(* Schneider Machine Expert - Basic project Sala de metrologia 174.3-2026 alteracao set umidade, file version 2.7.0.0 *)
(* CompanyInformations: Name=Kaefer - Mercedes Benz - Delma, PhoneNumber=11975904673, Street=RUA ALFRED JURZYKOWSKI 56, City=SÃO BERNARDO DO CAMPO, ZipCode=09680-900, State=SÃO PAULO, Country=BRASIL, WebSite=MERCEDES BENZ *)
(* ProjectInformations: Name=CLP DE CONTROLE METROLOGIA 21, Description=SUBSTITUIÇÃO DO CLP SPYDER PUB4024S DA FABRICANTE HONEYWELL COM AVÁRIA POR OUTRO DA FABRICANTE SCHNEIDER:

MODELO DA CPU: TM221ME 16T/MG COM EXPANSÃO DE SAIDA ANÁLOGICA: TM3AQ2 COM DUAS SAIDA ANÁLOGICAS;

O PROJETO CONSISTE EM MANTER A TEMPERATURA EM 19.5°C a 20.8°C E UMIDADE 45 A 55% *)

HARDWARE
  Cpu 0: TM221ME16T/G
  ModuleExtensionObject 0: TM3AQ2/G
  EthernetConfiguration: NetworkName=M221, IpAllocationMode=FixedAddress, IpAddress=192.168.1.5, SubnetMask=255.255.255.0
  SerialLineConfiguration: Baud=Baud19200, Parity=ParityEven, DataBits=DataBits8, StopBits=StopBits1, PhysicalMedium=PhysicalMediumRs485, TransmissionMode=TransmissionModeModbusRtu, SlaveId=1, Addressing=SlaveAddressing
  MastTask: UsePeriodScanMode=false, PeriodScan=100
  FastTask: Period=255
  CpuBehavior: StartingMode=StartAsPreviousState, AutoSaveRamOnEeprom=true, WatchdogPeriod=250

SYMBOLS  (address, symbol, comment, settings)
  %M0       HABILITA_GERAL_  "Memoria de habilita geral"
  %M1       COMP_1_LIGAR_  "habilita compressor 1"
  %M2       LIGA_COMP_2  "habilita compressor 2"
  %M4       LIGA_VENTILAÇÃO
  %M5       STATUS_VENT_LIGA
  %M6       HABILITA_AQUEC
  %M8       FOTO_CELULA
  %S6       SB_TB1S  "Base de tempo de 1 s gerada por um relógio interno"
  %I0.0       "Habilita geral"
  %I0.1     TERMOSTATO_DE_SEG
  %I0.2     STATUS_VENT
  %I0.3     CHAVE_DE_FLUXO_
  %I0.4     PRESSOSTATO
  %Q0.0     VENTILADOR_LIGA_DESLIGA
  %Q0.1     COMPRESSOR_1__LIGADO_
  %Q0.2     COMP_2_LIGAR_
  %Q0.3     LIGA_UMIDIFICAÇÃO_
  %Q0.4     INIBIÇÃO_AQUECIMENTO
  %IW0.0      [Type=Type_0_10V, Scope=Scope_Normal, Minimum=0, Maximum=1000]
  %IW0.1      [Type=Type_0_10V, Scope=Scope_Normal, Minimum=0, Maximum=1000]
  %QW1.0      [Type=Type_0_10V, Scope=Scope_Customized, Minimum=0, Maximum=10000]

POU Novo POU
  (* SectionNumber=1 *)

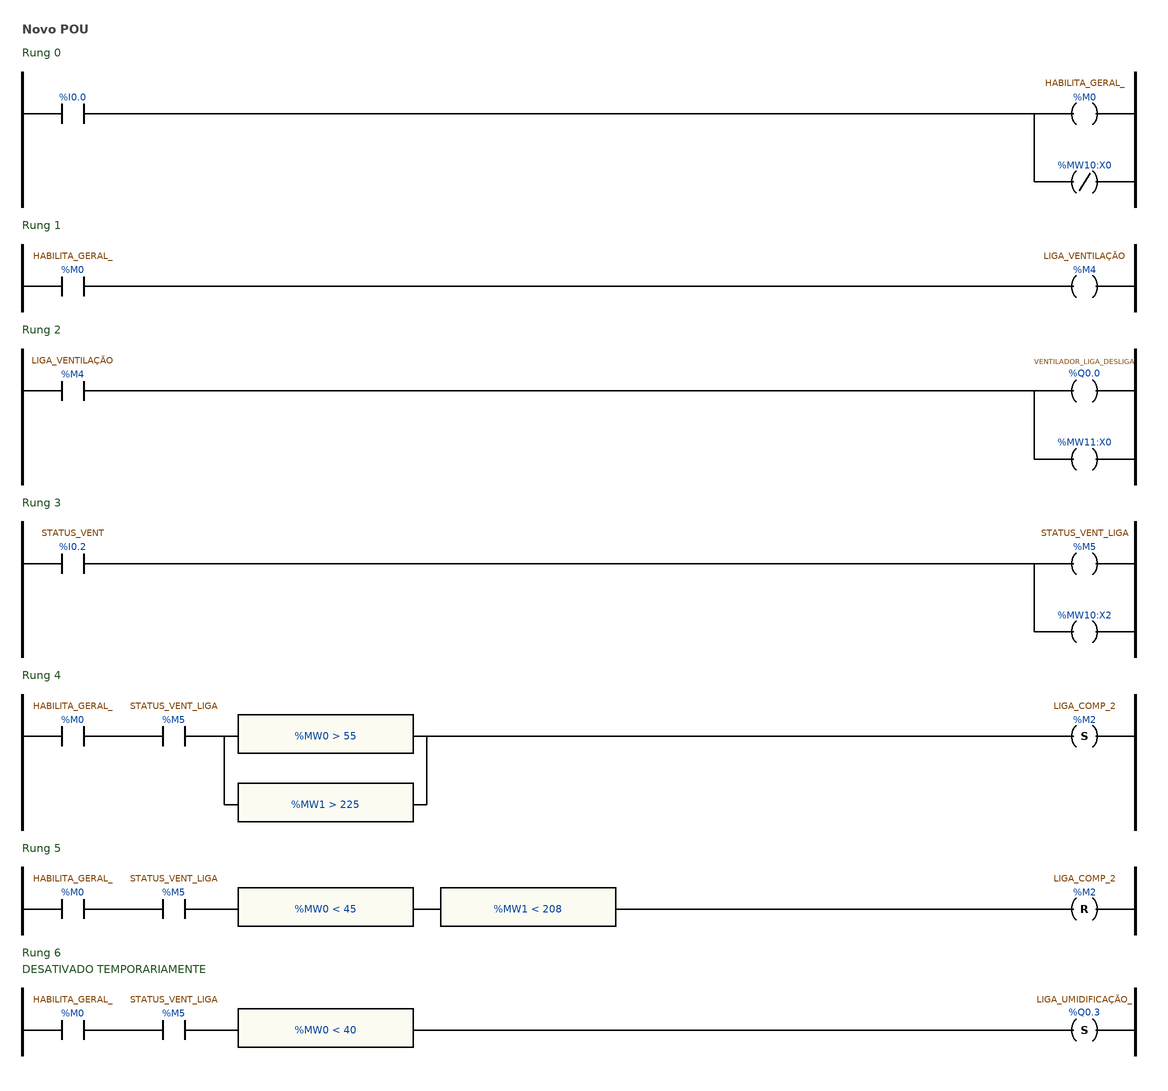

// Rung 0
  LD %I0.0
  ST %M0                  (* HABILITA_GERAL_ *)
  STN %MW10:X0
  // as ST:
  //   HABILITA_GERAL_ := %I0.0;
  //   %MW10:X0 := NOT %I0.0;

// Rung 1
  LD %M0                  (* HABILITA_GERAL_ *)
  ST %M4                  (* LIGA_VENTILAÇÃO *)
  // as ST:
  //   LIGA_VENTILAÇÃO := HABILITA_GERAL_;

// Rung 2
  LD %M4                  (* LIGA_VENTILAÇÃO *)
  ST %Q0.0                (* VENTILADOR_LIGA_DESLIGA *)
  ST %MW11:X0
  // as ST:
  //   VENTILADOR_LIGA_DESLIGA := LIGA_VENTILAÇÃO;
  //   %MW11:X0 := LIGA_VENTILAÇÃO;

// Rung 3
  LD %I0.2                (* STATUS_VENT *)
  ST %M5                  (* STATUS_VENT_LIGA *)
  ST %MW10:X2
  // as ST:
  //   STATUS_VENT_LIGA := STATUS_VENT;
  //   %MW10:X2 := STATUS_VENT;

// Rung 4
  LD %M0                  (* HABILITA_GERAL_ *)
  AND %M5                 (* STATUS_VENT_LIGA *)
  AND( [ %MW0 > 55 ]
  OR [ %MW1 > 225 ]
  )
  S %M2                   (* LIGA_COMP_2 *)
  // as ST:
  //   IF HABILITA_GERAL_ AND STATUS_VENT_LIGA AND (%MW0 > 55 OR %MW1 > 225) THEN LIGA_COMP_2 := TRUE; END_IF;

// Rung 5
  LD %M0                  (* HABILITA_GERAL_ *)
  AND %M5                 (* STATUS_VENT_LIGA *)
  AND [ %MW0 < 45 ]
  AND [ %MW1 < 208 ]
  R %M2                   (* LIGA_COMP_2 *)
  // as ST:
  //   IF HABILITA_GERAL_ AND STATUS_VENT_LIGA AND %MW0 < 45 AND %MW1 < 208 THEN LIGA_COMP_2 := FALSE; END_IF;

// Rung 6
// DESATIVADO TEMPORARIAMENTE
  LD %M0                  (* HABILITA_GERAL_ *)
  AND %M5                 (* STATUS_VENT_LIGA *)
  AND [ %MW0 < 40 ]
  S %Q0.3                 (* LIGA_UMIDIFICAÇÃO_ *)
  // as ST:
  //   IF HABILITA_GERAL_ AND STATUS_VENT_LIGA AND %MW0 < 40 THEN LIGA_UMIDIFICAÇÃO_ := TRUE; END_IF;

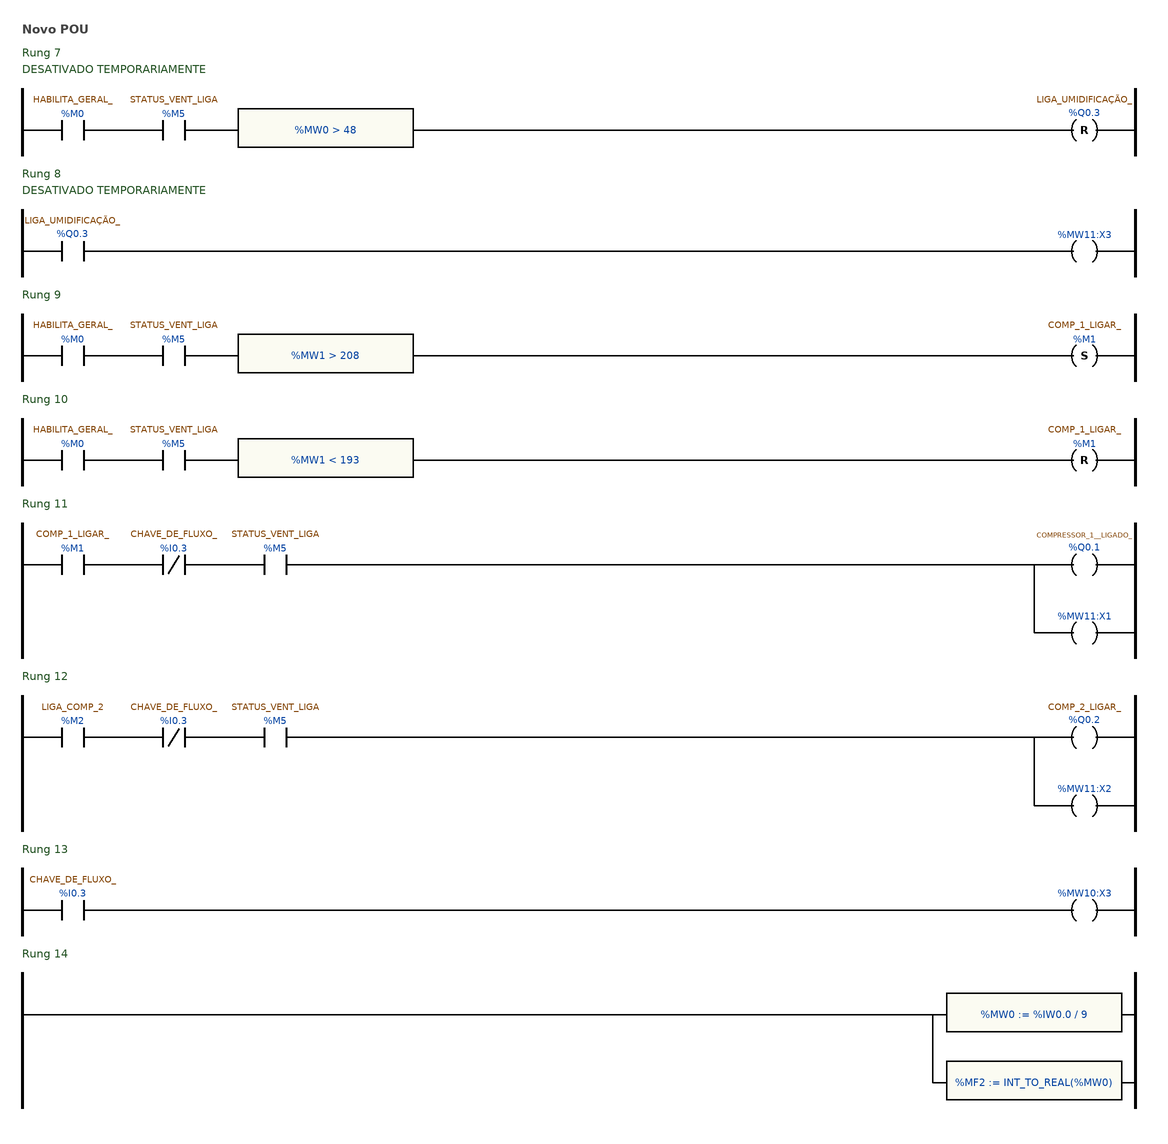

// Rung 7
// DESATIVADO TEMPORARIAMENTE
  LD %M0                  (* HABILITA_GERAL_ *)
  AND %M5                 (* STATUS_VENT_LIGA *)
  AND [ %MW0 > 48 ]
  R %Q0.3                 (* LIGA_UMIDIFICAÇÃO_ *)
  // as ST:
  //   IF HABILITA_GERAL_ AND STATUS_VENT_LIGA AND %MW0 > 48 THEN LIGA_UMIDIFICAÇÃO_ := FALSE; END_IF;

// Rung 8
// DESATIVADO TEMPORARIAMENTE
  LD %Q0.3                (* LIGA_UMIDIFICAÇÃO_ *)
  ST %MW11:X3
  // as ST:
  //   %MW11:X3 := LIGA_UMIDIFICAÇÃO_;

// Rung 9
  LD %M0                  (* HABILITA_GERAL_ *)
  AND %M5                 (* STATUS_VENT_LIGA *)
  AND [ %MW1 > 208 ]
  S %M1                   (* COMP_1_LIGAR_ *)
  // as ST:
  //   IF HABILITA_GERAL_ AND STATUS_VENT_LIGA AND %MW1 > 208 THEN COMP_1_LIGAR_ := TRUE; END_IF;

// Rung 10
  LD %M0                  (* HABILITA_GERAL_ *)
  AND %M5                 (* STATUS_VENT_LIGA *)
  AND [ %MW1 < 193 ]
  R %M1                   (* COMP_1_LIGAR_ *)
  // as ST:
  //   IF HABILITA_GERAL_ AND STATUS_VENT_LIGA AND %MW1 < 193 THEN COMP_1_LIGAR_ := FALSE; END_IF;

// Rung 11
  LD %M1                  (* COMP_1_LIGAR_ *)
  ANDN %I0.3              (* CHAVE_DE_FLUXO_ *)
  AND %M5                 (* STATUS_VENT_LIGA *)
  ST %Q0.1                (* COMPRESSOR_1__LIGADO_ *)
  ST %MW11:X1
  // as ST:
  //   COMPRESSOR_1__LIGADO_ := COMP_1_LIGAR_ AND NOT CHAVE_DE_FLUXO_ AND STATUS_VENT_LIGA;
  //   %MW11:X1 := COMP_1_LIGAR_ AND NOT CHAVE_DE_FLUXO_ AND STATUS_VENT_LIGA;

// Rung 12
  LD %M2                  (* LIGA_COMP_2 *)
  ANDN %I0.3              (* CHAVE_DE_FLUXO_ *)
  AND %M5                 (* STATUS_VENT_LIGA *)
  ST %Q0.2                (* COMP_2_LIGAR_ *)
  ST %MW11:X2
  // as ST:
  //   COMP_2_LIGAR_ := LIGA_COMP_2 AND NOT CHAVE_DE_FLUXO_ AND STATUS_VENT_LIGA;
  //   %MW11:X2 := LIGA_COMP_2 AND NOT CHAVE_DE_FLUXO_ AND STATUS_VENT_LIGA;

// Rung 13
  LD %I0.3                (* CHAVE_DE_FLUXO_ *)
  ST %MW10:X3
  // as ST:
  //   %MW10:X3 := CHAVE_DE_FLUXO_;

// Rung 14
  LD 1
  [ %MW0 := %IW0.0 / 9 ]
  [ %MF2 := INT_TO_REAL ( %MW0 ) ]
  // as ST:
  //   %MW0 := %IW0.0 / 9;
  //   %MF2 := INT_TO_REAL ( %MW0 );

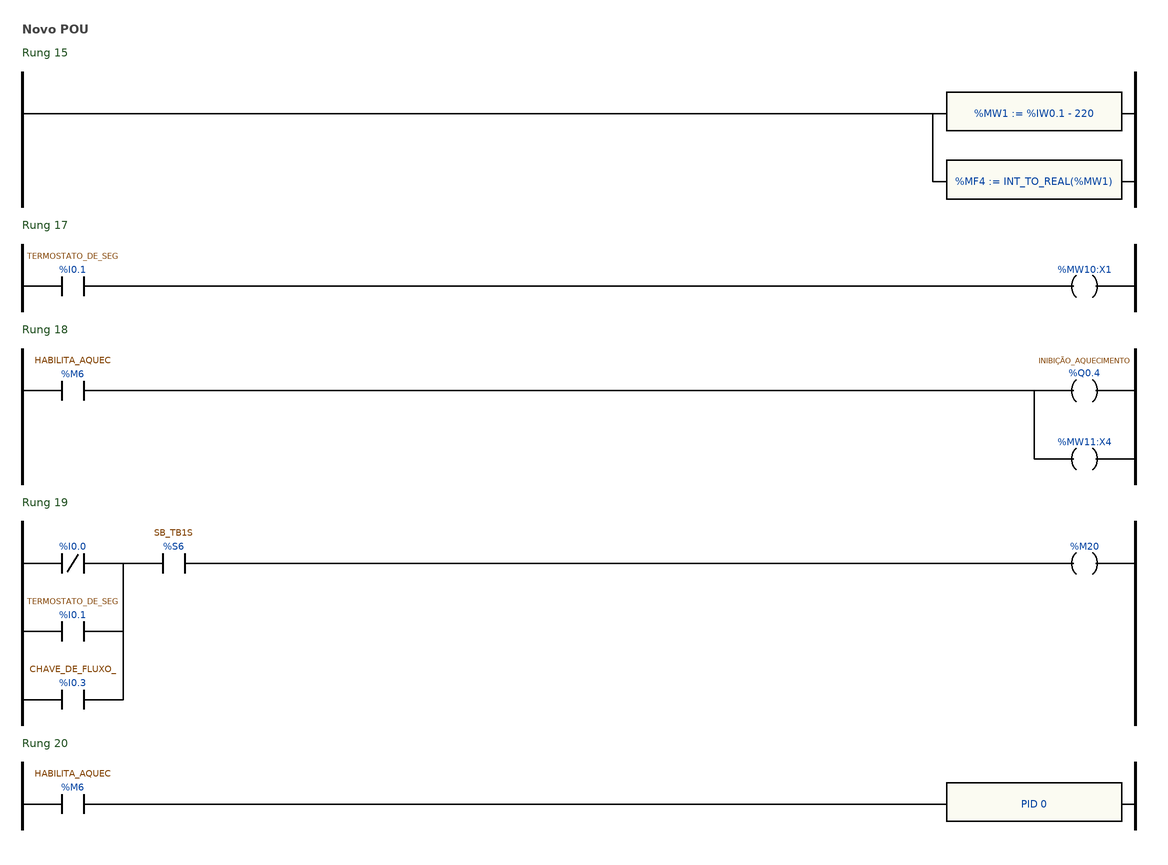

// Rung 15
  LD 1
  [ %MW1 := %IW0.1 - 220 ]
  [ %MF4 := INT_TO_REAL ( %MW1 ) ]
  // as ST:
  //   %MW1 := %IW0.1 - 220;
  //   %MF4 := INT_TO_REAL ( %MW1 );

// Rung 16
  LD %M5                  (* STATUS_VENT_LIGA *)
  ANDN %I0.1              (* TERMOSTATO_DE_SEG *)
  ANDN %I0.3              (* CHAVE_DE_FLUXO_ *)
  AND [ %MW1 > 225 ]
  ST %M6                  (* HABILITA_AQUEC *)
  // as ST:
  //   HABILITA_AQUEC := STATUS_VENT_LIGA AND NOT TERMOSTATO_DE_SEG AND NOT CHAVE_DE_FLUXO_ AND %MW1 > 225;
  (* the ladder stored for this rung does not match its IL; not drawn *)

// Rung 17
  LD %I0.1                (* TERMOSTATO_DE_SEG *)
  ST %MW10:X1
  // as ST:
  //   %MW10:X1 := TERMOSTATO_DE_SEG;

// Rung 18
  LD %M6                  (* HABILITA_AQUEC *)
  ST %Q0.4                (* INIBIÇÃO_AQUECIMENTO *)
  ST %MW11:X4
  // as ST:
  //   INIBIÇÃO_AQUECIMENTO := HABILITA_AQUEC;
  //   %MW11:X4 := HABILITA_AQUEC;

// Rung 19
  LDN %I0.0
  OR %I0.1                (* TERMOSTATO_DE_SEG *)
  OR %I0.3                (* CHAVE_DE_FLUXO_ *)
  AND %S6                 (* SB_TB1S *)
  ST %M20
  // as ST:
  //   %M20 := (NOT %I0.0 OR TERMOSTATO_DE_SEG OR CHAVE_DE_FLUXO_) AND SB_TB1S;

// Rung 20
  LD %M6                  (* HABILITA_AQUEC *)
  [ PID 0 ]
  // as ST:
  //   IF HABILITA_AQUEC THEN PID 0; END_IF;

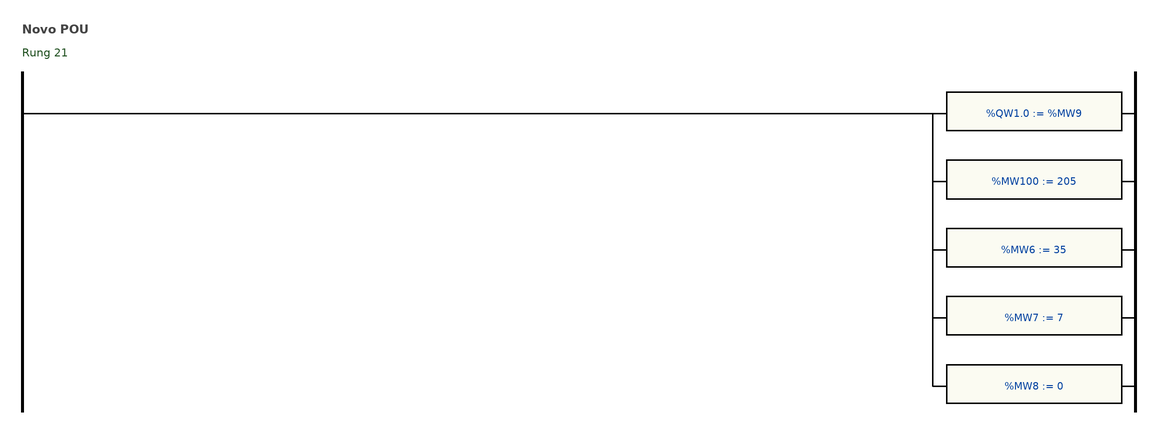

// Rung 21
  LD 1
  [ %QW1.0 := %MW9 ]
  [ %MW100 := 205 ]
  [ %MW6 := 35 ]
  [ %MW7 := 7 ]
  [ %MW8 := 0 ]
  // as ST:
  //   %QW1.0 := %MW9;
  //   %MW100 := 205;
  //   %MW6 := 35;
  //   %MW7 := 7;
  //   %MW8 := 0;
